// TIA Portal project "260113_Aufgabe_03" (V20)

(* hardware
DEVICE "S7-300/ET200M-Station_1"  S7-300 station
   slot 0: "Profilschiene_0"  Rail  6ES7 390-1***0-0AA0
   slot 2: "PLC_1"  CPU 315-2 PN/DP  6ES7 315-2EH14-0AB0  V3.2.18
      slot 2: "PROFINET-Schnittstelle_1"  PN-IO
         slot 1: "Port_1"  Port
         slot 2: "Port_2"  Port
   slot 4: "DI 16x24VDC_1"  DI16 x 24VDC, interrupt  6ES7 321-7BH01-0AB0
   slot 5: "DO 16x24VDC/0.5A_1"  DO16xDC24V/0.5A  6ES7 322-8BH10-0AB0
   slot 6: "DI 16x24VDC_2"  DI16 x 24VDC, interrupt  6ES7 321-7BH01-0AB0
   slot 7: "DO 16x24VDC/0.5A_2"  DO16xDC24V/0.5A  6ES7 322-8BH10-0AB0
   slot 8: "DI 64x24VDC Sinking/Sourcing_1"  DI64 x 24VDC  6ES7 321-1BP00-0AA0
   slot 9: "DO 64x24VDC/0.3A sinking_1"  DO64 x 24VDC / 0.3A, M  6ES7 322-1BP50-0AA0
*)

// ===== PLC "PLC_1"  CPU 315-2 PN/DP =====

VAR_GLOBAL   // PLC tag table "Standard-Variablentabelle"
   "100Hz_Takt" AT %M100.5 : Bool;
END_VAR

VAR_GLOBAL   // PLC tag table "Abfüllanlagen-Tabelle"
   "Vorratsbehälter_1" AT %E0.0 : Bool;
   "Vorratsbehälter_2" AT %E0.1 : Bool;
   "Warnlicht_1" AT %A0.0 : Bool;
   "Warnlicht_2" AT %A0.1 : Bool;
   "Motor_0" AT %A0.4 : Bool;
   "Vorratsbehälter_1_leer" AT %M0.0 : Bool;
   "Vorratsbehälter_2_leer" AT %M0.1 : Bool;
END_VAR

VAR_GLOBAL   // PLC tag table "Bustüren-Tabelle"
   "Tür_1" AT %E1.0 : Bool;
   "Tür_2" AT %E1.1 : Bool;
   "Tür_3" AT %E1.2 : Bool;
   "Signallampe_0" AT %A1.0 : Bool;
   "Tür_1_offen" AT %M1.0 : Bool;
   "Tür_2_offen" AT %M1.1 : Bool;
   "Tür_3_offen" AT %M1.2 : Bool;
END_VAR

VAR_GLOBAL   // PLC tag table "Temperaturü.-Tabelle"
   "Sensor_1" AT %E2.0 : Bool;
   "Sensor_2" AT %E2.1 : Bool;
   "Sensor_3" AT %E2.2 : Bool;
   "Sensor_4" AT %E2.3 : Bool;
   "Rücksetztaster" AT %E2.4 : Bool;
   "Anzeige_0" AT %A2.0 : Bool;
END_VAR

VAR_GLOBAL   // PLC tag table "Hausbeleuchtung-Tabelle"
   "Helligkeitssensor" AT %E3.0 : Bool;
   "Bewegungssensor" AT %E3.1 : Bool;
   "Handbetrieb" AT %E3.2 : Bool;
   "Beleuchtung" AT %A3.0 : Bool;
END_VAR

VAR_GLOBAL   // PLC tag table "Not-Aus_Förderband-Tabelle"
   "Bandtaster_1" AT %E4.0 : Bool;
   "Bandtaster_2" AT %E4.1 : Bool;
   "Lichtschranke" AT %E4.4 : Bool;
   "Not-Aus zurücksetzen" AT %E4.5 : Bool;
   "Förderband" AT %A4.0 : Bool;
   "Förderband aktiv" AT %M4.0 : Bool;
   "Not-Aus aktiv" AT %M4.1 : Bool;
END_VAR

VAR_GLOBAL   // PLC tag table "Quizshow-Tabelle"
   "Teilnehmer_1" AT %E5.0 : Bool;
   "Teilnehmer_2" AT %E5.1 : Bool;
   "Moderator Freigabe" AT %E5.7 : Bool;
   "TN_1-Lampe" AT %A5.0 : Bool;
   "TN_2-Lampe" AT %A5.1 : Bool;
   "TN_1-Gedrückt" AT %M5.0 : Bool;
   "TN_2-Gedrückt" AT %M5.1 : Bool;
   "Freigabe erteilt" AT %M5.7 : Bool;
END_VAR

VAR_GLOBAL   // PLC tag table "Pförtnerschranke-Tabelle"
   "Sperre" AT %E6.0 : Bool;
   "Knopf hoch" AT %E6.1 : Bool;
   "Knopf runter" AT %E6.2 : Bool;
   "Schrankenmotor vorwärts" AT %A6.0 : Bool;
   "Schrankenmotor rückwärts" AT %A6.1 : Bool;
   "Rotes_Signal_0" AT %A6.2 : Bool;
   "Schranke fährt hoch" AT %M6.0 : Bool;
   "Schranke fährt runter" AT %M6.1 : Bool;
END_VAR

FUNCTION_BLOCK "Abfüllanlage"   // FB1, FBD
{ S7_Optimized_Access := 'FALSE' }
VERSION : 0.1
BEGIN

REGION Network 1: Behältersteuerung 1
   // Die Warnleuchte geht an, sobald der Behälter zu wenig Inhalt hat.
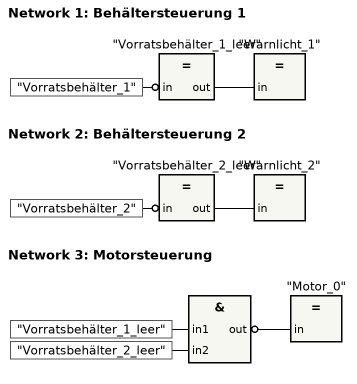
   "Vorratsbehälter_1_leer" := NOT "Vorratsbehälter_1";
   "Warnlicht_1" := NOT "Vorratsbehälter_1";
END_REGION

REGION Network 2: Behältersteuerung 2
   // Die Warnleuchte geht an, sobald der Behälter zu wenig Inhalt hat.
   "Vorratsbehälter_2_leer" := NOT "Vorratsbehälter_2";
   "Warnlicht_2" := NOT "Vorratsbehälter_2";
END_REGION

REGION Network 3: Motorsteuerung
   // Der Motor wird abgeschaltet, sobald beide Behälter leer sind. Ansonsten ist dieser aktiv.
   "Motor_0" := NOT ("Vorratsbehälter_1_leer" AND "Vorratsbehälter_2_leer");
END_REGION
END_FUNCTION_BLOCK

FUNCTION_BLOCK "Bustüren"   // FB2, FBD
{ S7_Optimized_Access := 'FALSE' }
VERSION : 0.1
BEGIN

REGION Network 1: Bustür
   // Siehe Netzwerk 3.
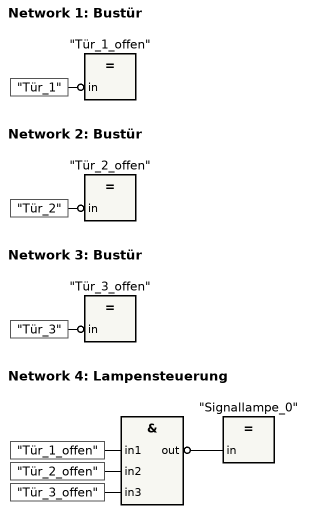
   "Tür_1_offen" := NOT "Tür_1";
END_REGION

REGION Network 2: Bustür
   // Siehe Netzwerk 3.
   "Tür_2_offen" := NOT "Tür_2";
END_REGION

REGION Network 3: Bustür
   // Jede Bustür bekommt einen Merker. Wenn Strom anliegt ist die Tür offen, ansonsten geschlossen.
   "Tür_3_offen" := NOT "Tür_3";
END_REGION

REGION Network 4: Lampensteuerung
   // Die Signallampe geht aus wenn alle Türen geschlossen sind.
   "Signallampe_0" := NOT ("Tür_1_offen" AND "Tür_2_offen" AND "Tür_3_offen");
END_REGION
END_FUNCTION_BLOCK

FUNCTION_BLOCK "Temperaturüberwachung"   // FB3, FBD
{ S7_Optimized_Access := 'FALSE' }
VERSION : 0.1
BEGIN

REGION Network 1: Überwachungssteuerung
   // Wenn einer der Sensoren etwas meldet, geht die Anzeige an. Wenn das Problem dann behoben wurde, also kein Sensor mehr etwas meldet, kann mit dem Rücksetztaster die Anzeige zurückgesetzt werden.
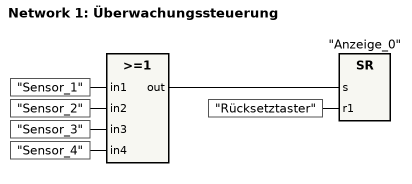
   IF "Sensor_1" OR "Sensor_2" OR "Sensor_3" OR "Sensor_4" THEN
       "Anzeige_0" := TRUE;   // SR flip-flop
   END_IF;
   IF "Rücksetztaster" THEN "Anzeige_0" := FALSE; END_IF;
END_REGION
END_FUNCTION_BLOCK

FUNCTION_BLOCK "Hausbeleuchtung"   // FB4, FBD
{ S7_Optimized_Access := 'FALSE' }
VERSION : 0.1
BEGIN

REGION Network 1: Haus-Außenbeleuchtung
   // Sobald es dunkel ist und der Bewegungsmelder eine Person oder ein Auto wahnimmt, geht die Beleuchtung an. Die Beleuchtung kann aber auch manuell mit Handbetrieb an-/ausgeschaltet werden.
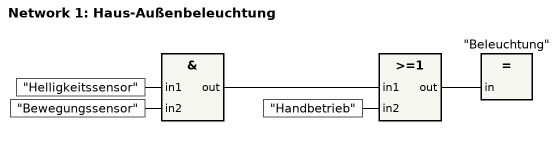
   "Beleuchtung" := ("Helligkeitssensor" AND "Bewegungssensor") OR "Handbetrieb";
END_REGION
END_FUNCTION_BLOCK

FUNCTION_BLOCK "Not-Aus_Förderband"   // FB5, FBD
{ S7_Optimized_Access := 'FALSE' }
VERSION : 0.1
BEGIN

REGION Network 1: Förderbandsteuerung
   // Solange beide Taster gedrückt sind, läuft das Förderband. Wenn die Lichtschranke ein Signal sendet, dann ist der Not-Aus aktiv und das Förderband bleibt gestoppt. Nun muss der Not-Aus zurückgesetzt werden, damit das Förderband weiterläuft.
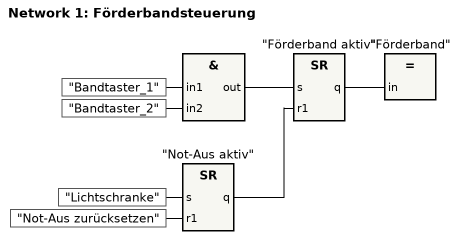
   IF "Lichtschranke" THEN
       "Not-Aus aktiv" := TRUE;   // SR flip-flop
   END_IF;
   IF "Not-Aus zurücksetzen" THEN "Not-Aus aktiv" := FALSE; END_IF;
   IF "Bandtaster_1" AND "Bandtaster_2" THEN
       "Förderband aktiv" := TRUE;   // SR flip-flop
   END_IF;
   IF "Not-Aus aktiv" THEN "Förderband aktiv" := FALSE; END_IF;
   "Förderband" := "Förderband aktiv";
END_REGION
END_FUNCTION_BLOCK

FUNCTION_BLOCK "Quizshow"   // FB6, FBD
{ S7_Optimized_Access := 'FALSE' }
VERSION : 0.1
BEGIN

REGION Network 1: Teilnehmerbuzzer
   // Siehe Netzwerk 2.
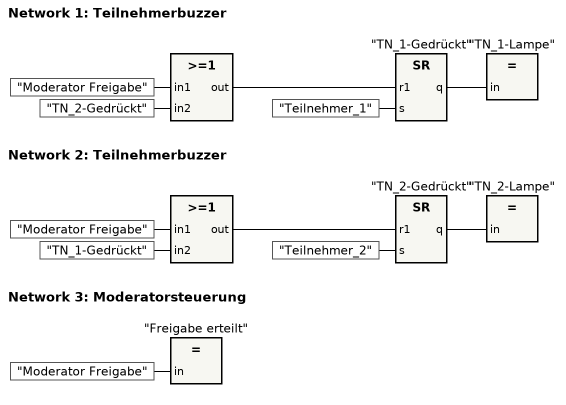
   IF "Teilnehmer_1" THEN
       "TN_1-Gedrückt" := TRUE;   // SR flip-flop
   END_IF;
   IF "Moderator Freigabe" OR "TN_2-Gedrückt" THEN "TN_1-Gedrückt" := FALSE; END_IF;
   "TN_1-Lampe" := "TN_1-Gedrückt";
END_REGION

REGION Network 2: Teilnehmerbuzzer
   // Sobald der andere Teilnehmer buzzert, wird der Buzzer für diesen Teilnehmer gesperrt. Sollte dieser Teilnehmer zuerst Buzzern ist es genau umgekehrt und zusätzlich geht die Lampe dieses Teilnehmers an. Der Moderator kann den Buzzer für diesen Teilnehmer sperren und (wieder) frei geben.
   IF "Teilnehmer_2" THEN
       "TN_2-Gedrückt" := TRUE;   // SR flip-flop
   END_IF;
   IF "Moderator Freigabe" OR "TN_1-Gedrückt" THEN "TN_2-Gedrückt" := FALSE; END_IF;
   "TN_2-Lampe" := "TN_2-Gedrückt";
END_REGION

REGION Network 3: Moderatorsteuerung
   // Der Moderator kann die Buzzer der Teilnehmer sperren und wieder frei geben.
   "Freigabe erteilt" := "Moderator Freigabe";
END_REGION
END_FUNCTION_BLOCK

FUNCTION_BLOCK "Pförtnerschranke"   // FB7, FBD
{ S7_Optimized_Access := 'FALSE' }
VERSION : 0.1
BEGIN

REGION Network 1: Schrankensteuerung Hoch
   // Siehe Netzwerk 2.
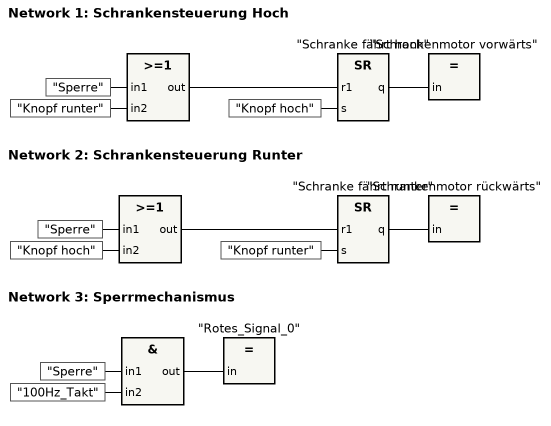
   IF "Knopf hoch" THEN
       "Schranke fährt hoch" := TRUE;   // SR flip-flop
   END_IF;
   IF "Sperre" OR "Knopf runter" THEN "Schranke fährt hoch" := FALSE; END_IF;
   "Schrankenmotor vorwärts" := "Schranke fährt hoch";
END_REGION

REGION Network 2: Schrankensteuerung Runter
   // Wenn die Sperre aktiv ist oder der andere Knopf gerade betätigt wird, kann dieser Knopf nicht betätigt werden. Sind die beiden Bedingungen nicht gegeben, wird über den Knopf der Schrankenmotor in eine Richtung gesteuert.
   IF "Knopf runter" THEN
       "Schranke fährt runter" := TRUE;   // SR flip-flop
   END_IF;
   IF "Sperre" OR "Knopf hoch" THEN "Schranke fährt runter" := FALSE; END_IF;
   "Schrankenmotor rückwärts" := "Schranke fährt runter";
END_REGION

REGION Network 3: Sperrmechanismus
   // Sobald der Pförtner seinen Arbeitsplatz verlässt, blinkt die rote Signalleuchte, die Sperre ist aktiv.
   "Rotes_Signal_0" := "Sperre" AND "100Hz_Takt";
END_REGION
END_FUNCTION_BLOCK

ORGANIZATION_BLOCK "Main"   // OB1, FBD
TITLE = "Main Program Sweep (Cycle)"
{ S7_Optimized_Access := 'FALSE' }
VERSION : 0.1
   VAR_TEMP
      OB1_EV_CLASS : Byte;   // Bits 0-3 = 1 (Coming event), Bits 4-7 = 1 (Event class 1)
      OB1_SCAN_1 : Byte;   // 1 (Cold restart scan 1 of OB 1), 3 (Scan 2-n of OB 1)
      OB1_PRIORITY : Byte;   // Priority of OB Execution
      OB1_OB_NUMBR : Byte;   // 1 (Organization block 1, OB1)
      OB1_RESERVED_1 : Byte;   // Reserved for system
      OB1_RESERVED_2 : Byte;   // Reserved for system
      OB1_PREV_CYCLE : Int;   // Cycle time of previous OB1 scan (milliseconds)
      OB1_MIN_CYCLE : Int;   // Minimum cycle time of OB1 (milliseconds)
      OB1_MAX_CYCLE : Int;   // Maximum cycle time of OB1 (milliseconds)
      OB1_DATE_TIME : Date_And_Time;   // Date and time OB1 started
   END_VAR
BEGIN
END_ORGANIZATION_BLOCK